Omron Sysmac Studio project SPA_P6 (Sysmac Studio 1.23.0.14, StandardProject)

# Controller new_Controller_0: NX1P2-1040DT1 version 1.18
Task PrimaryTask (priority 4, period or condition 2000): Programa0

VAR_GLOBAL
    PM : BOOL;  (* Pulsador de Marcha; at BuiltInIO://cpu/#0/Input_Bit_00 *)
    PP : BOOL;  (* Pulsador de Paro; at BuiltInIO://cpu/#0/Input_Bit_01 *)
    O0 : BOOL;  (* Salida 0; at BuiltInIO://cpu/#0/Output_Bit_00 *)
    HMI_PM AT %W0.0 : BOOL;  (* published *)
    HMI_PP AT %W0.1 : BOOL;  (* published *)
END_VAR
VAR_GLOBAL RETAIN
    out_number AT %D0 : REAL;  (* published *)
    in_number AT %D2 : INT;  (* published *)
END_VAR
VAR_GLOBAL
    O2 : BOOL;  (* at BuiltInIO://cpu/#0/Output_Bit_02 *)
END_VAR

PROGRAM Programa0
VAR
    hmi : BOOL;
    working : BOOL;
    variable : BOOL;
END_VAR
VAR_EXTERNAL
    PM : BOOL;
    PP : BOOL;
    O0 : BOOL;
    HMI_PM : BOOL;
    HMI_PP : BOOL;
    O2 : BOOL;
    in_number : INT;
    out_number : REAL;
END_VAR

(* Section Sección0: ladder, written here as Structured Text *)

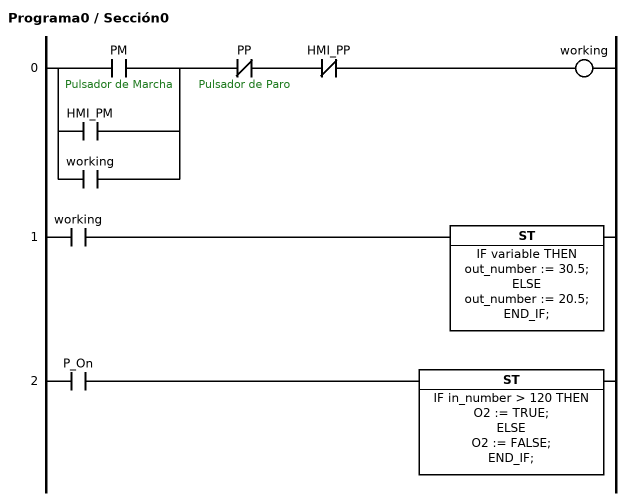
(* Rung 0 *)
working := (PM OR HMI_PM OR working) AND NOT PP AND NOT HMI_PP;
(* Rung 1 *)
IF working THEN
    IF variable THEN
         out_number := 30.5;
    ELSE
         out_number := 20.5;
    END_IF;
END_IF;
(* Rung 2 *)
IF P_On THEN
    IF in_number > 120 THEN
         O2 := TRUE;
    ELSE
         O2 := FALSE;
    END_IF;
END_IF;
END_PROGRAM